SYSTEM Test System
  (* Version 1.0, 2005-06-15, Goran Cengic, Chalmers *)
  DEVICE Test Device : DeviceType_not_used
    RESOURCE Test Resource : ResourceType_not_used
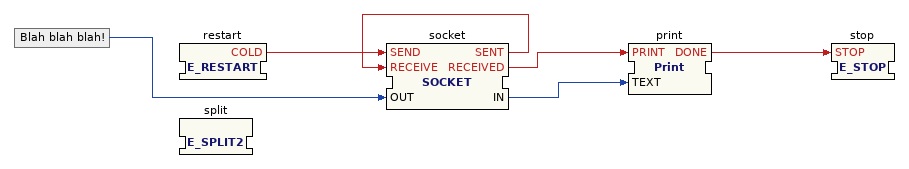
      FBS
        restart : E_RESTART;
        split : E_SPLIT2;
        socket : SOCKET;
        print : Print;
        stop : E_STOP;
      END_FBS
      EVENT_CONNECTIONS
        restart.COLD TO socket.SEND;
        socket.SENT TO socket.RECEIVE;
        socket.RECEIVED TO print.PRINT;
        print.DONE TO stop.STOP;
      END_CONNECTIONS
      DATA_CONNECTIONS
        Blah blah blah! TO socket.OUT;
        socket.IN TO print.TEXT;
      END_CONNECTIONS
    END_RESOURCE
  END_DEVICE
END_SYSTEM
